# EPICS substitutions: db/MLout.substitutions
file "/epics/iocs/MachineLearn/db/MLout_sub.db"
{
pattern
{CELL, WIRE,  MODE}
{"01", "33", "lls"}
{"01", "34", "lls"}
{"01", "35", "lls"}
{"01", "36", "lls"}
{"01", "37", "lls"}
{"01", "38", "lls"}
{"01", "39", "lls"}
{"01", "40", "lls"}
{"01", "41", "lls"}
{"01", "42", "lls"}
{"01", "43", "lls"}
{"01", "44", "lls"}
{"01", "45", "lls"}
{"01", "46", "lls"}
{"01", "47", "lls"}
{"01", "48", "lls"}
{"01", "49", "lls"}
{"01", "50", "lls"}
{"01", "51", "lls"}
{"01", "52", "lls"}

{"02", "33", "lls"}
{"02", "34", "lls"}
{"02", "35", "lls"}
{"02", "36", "lls"}
{"02", "37", "lls"}
{"02", "38", "lls"}
{"02", "39", "lls"}
{"02", "40", "lls"}
{"02", "41", "lls"}
{"02", "42", "lls"}
{"02", "43", "lls"}
{"02", "44", "lls"}
{"02", "45", "lls"}
{"02", "46", "lls"}
{"02", "47", "lls"}
{"02", "48", "lls"}
{"02", "49", "lls"}
{"02", "50", "lls"}
{"02", "51", "lls"}
{"02", "52", "lls"}

{"03", "55", "lls"}
{"03", "56", "lls"}
{"03", "57", "lls"}
{"03", "58", "lls"}
{"03", "59", "lls"}
{"03", "60", "lls"}
{"03", "61", "lls"}
{"03", "62", "lls"}
{"03", "63", "lls"}
{"03", "64", "lls"}
{"03", "65", "lls"}
{"03", "66", "lls"}
{"03", "67", "lls"}
{"03", "68", "lls"}
{"03", "69", "lls"}
{"03", "70", "lls"}
{"03", "71", "lls"}
{"03", "72", "lls"}
{"03", "73", "lls"}
{"03", "74", "lls"}

{"04", "33", "lls"}
{"04", "34", "lls"}
{"04", "35", "lls"}
{"04", "36", "lls"}
{"04", "37", "lls"}
{"04", "38", "lls"}
{"04", "39", "lls"}
{"04", "40", "lls"}
{"04", "41", "lls"}
{"04", "42", "lls"}
{"04", "43", "lls"}
{"04", "44", "lls"}
{"04", "45", "lls"}
{"04", "46", "lls"}
{"04", "47", "lls"}
{"04", "48", "lls"}
{"04", "49", "lls"}
{"04", "50", "lls"}
{"04", "51", "lls"}
{"04", "52", "lls"}

{"05", "33", "lls"}
{"05", "34", "lls"}
{"05", "35", "lls"}
{"05", "36", "lls"}
{"05", "37", "lls"}
{"05", "38", "lls"}
{"05", "39", "lls"}
{"05", "40", "lls"}
{"05", "41", "lls"}
{"05", "42", "lls"}
{"05", "43", "lls"}
{"05", "44", "lls"}
{"05", "45", "lls"}
{"05", "46", "lls"}
{"05", "47", "lls"}
{"05", "48", "lls"}
{"05", "49", "lls"}
{"05", "50", "lls"}
{"05", "51", "lls"}
{"05", "52", "lls"}

{"06", "33", "lls"}
{"06", "34", "lls"}
{"06", "35", "lls"}
{"06", "36", "lls"}
{"06", "37", "lls"}
{"06", "38", "lls"}
{"06", "39", "lls"}
{"06", "40", "lls"}
{"06", "41", "lls"}
{"06", "42", "lls"}
{"06", "43", "lls"}
{"06", "44", "lls"}
{"06", "45", "lls"}
{"06", "46", "lls"}
{"06", "47", "lls"}
{"06", "48", "lls"}
{"06", "49", "lls"}
{"06", "50", "lls"}
{"06", "51", "lls"}
{"06", "52", "lls"}

{"07", "33", "lls"}
{"07", "34", "lls"}
{"07", "35", "lls"}
{"07", "36", "lls"}
{"07", "37", "lls"}
{"07", "38", "lls"}
{"07", "39", "lls"}
{"07", "40", "lls"}
{"07", "41", "lls"}
{"07", "42", "lls"}
{"07", "43", "lls"}
{"07", "44", "lls"}
{"07", "45", "lls"}
{"07", "46", "lls"}
{"07", "47", "lls"}
{"07", "48", "lls"}
{"07", "49", "lls"}
{"07", "50", "lls"}
{"07", "51", "lls"}
{"07", "52", "lls"}

{"08", "33", "lls"}
{"08", "34", "lls"}
{"08", "35", "lls"}
{"08", "36", "lls"}
{"08", "37", "lls"}
{"08", "38", "lls"}
{"08", "39", "lls"}
{"08", "40", "lls"}
{"08", "41", "lls"}
{"08", "42", "lls"}
{"08", "43", "lls"}
{"08", "44", "lls"}
{"08", "45", "lls"}
{"08", "46", "lls"}
{"08", "47", "lls"}
{"08", "48", "lls"}
{"08", "49", "lls"}
{"08", "50", "lls"}
{"08", "51", "lls"}
{"08", "52", "lls"}

{"09", "33", "lls"}
{"09", "34", "lls"}
{"09", "35", "lls"}
{"09", "36", "lls"}
{"09", "37", "lls"}
{"09", "38", "lls"}
{"09", "39", "lls"}
{"09", "40", "lls"}
{"09", "41", "lls"}
{"09", "42", "lls"}
{"09", "43", "lls"}
{"09", "44", "lls"}
{"09", "45", "lls"}
{"09", "46", "lls"}
{"09", "47", "lls"}
{"09", "48", "lls"}
{"09", "49", "lls"}
{"09", "50", "lls"}
{"09", "51", "lls"}
{"09", "52", "lls"}

{"10", "33", "lls"}
{"10", "34", "lls"}
{"10", "35", "lls"}
{"10", "36", "lls"}
{"10", "37", "lls"}
{"10", "38", "lls"}
{"10", "39", "lls"}
{"10", "40", "lls"}
{"10", "41", "lls"}
{"10", "42", "lls"}
{"10", "43", "lls"}
{"10", "44", "lls"}
{"10", "45", "lls"}
{"10", "46", "lls"}
{"10", "47", "lls"}
{"10", "48", "lls"}
{"10", "49", "lls"}
{"10", "50", "lls"}
{"10", "51", "lls"}
{"10", "52", "lls"}

{"11", "33", "lls"}
{"11", "34", "lls"}
{"11", "35", "lls"}
{"11", "36", "lls"}
{"11", "37", "lls"}
{"11", "38", "lls"}
{"11", "39", "lls"}
{"11", "40", "lls"}
{"11", "41", "lls"}
{"11", "42", "lls"}
{"11", "43", "lls"}
{"11", "44", "lls"}
{"11", "45", "lls"}
{"11", "46", "lls"}
{"11", "47", "lls"}
{"11", "48", "lls"}
{"11", "49", "lls"}
{"11", "50", "lls"}
{"11", "51", "lls"}
{"11", "52", "lls"}

{"12", "33", "lls"}
{"12", "34", "lls"}
{"12", "35", "lls"}
{"12", "36", "lls"}
{"12", "37", "lls"}
{"12", "38", "lls"}
{"12", "39", "lls"}
{"12", "40", "lls"}
{"12", "41", "lls"}
{"12", "42", "lls"}
{"12", "43", "lls"}
{"12", "44", "lls"}
{"12", "45", "lls"}
{"12", "46", "lls"}
{"12", "47", "lls"}
{"12", "48", "lls"}
{"12", "49", "lls"}
{"12", "50", "lls"}
{"12", "51", "lls"}
{"12", "52", "lls"}

{"13", "33", "lls"}
{"13", "34", "lls"}
{"13", "35", "lls"}
{"13", "36", "lls"}
{"13", "37", "lls"}
{"13", "38", "lls"}
{"13", "39", "lls"}
{"13", "40", "lls"}
{"13", "41", "lls"}
{"13", "42", "lls"}
{"13", "43", "lls"}
{"13", "44", "lls"}
{"13", "45", "lls"}
{"13", "46", "lls"}
{"13", "47", "lls"}
{"13", "48", "lls"}
{"13", "49", "lls"}
{"13", "50", "lls"}
{"13", "51", "lls"}
{"13", "52", "lls"}
{"13", "53", "lls"}
{"13", "54", "lls"}
{"13", "55", "lls"}
{"13", "56", "lls"}

{"14", "33", "lls"}
{"14", "34", "lls"}
{"14", "35", "lls"}
{"14", "36", "lls"}
{"14", "37", "lls"}
{"14", "38", "lls"}
{"14", "39", "lls"}
{"14", "40", "lls"}
{"14", "41", "lls"}
{"14", "42", "lls"}
{"14", "43", "lls"}
{"14", "44", "lls"}
{"14", "45", "lls"}
{"14", "46", "lls"}
{"14", "47", "lls"}
{"14", "48", "lls"}
{"14", "49", "lls"}
{"14", "50", "lls"}
{"14", "51", "lls"}
{"14", "52", "lls"}

{"15", "33", "lls"}
{"15", "34", "lls"}
{"15", "35", "lls"}
{"15", "36", "lls"}
{"15", "37", "lls"}
{"15", "38", "lls"}
{"15", "39", "lls"}
{"15", "40", "lls"}
{"15", "41", "lls"}
{"15", "42", "lls"}
{"15", "43", "lls"}
{"15", "44", "lls"}
{"15", "45", "lls"}
{"15", "46", "lls"}
{"15", "47", "lls"}
{"15", "48", "lls"}
{"15", "49", "lls"}
{"15", "50", "lls"}
{"15", "51", "lls"}
{"15", "52", "lls"}

{"16", "33", "lls"}
{"16", "34", "lls"}
{"16", "35", "lls"}
{"16", "36", "lls"}
{"16", "37", "lls"}
{"16", "38", "lls"}
{"16", "39", "lls"}
{"16", "40", "lls"}
{"16", "41", "lls"}
{"16", "42", "lls"}
{"16", "43", "lls"}
{"16", "44", "lls"}
{"16", "45", "lls"}
{"16", "46", "lls"}
{"16", "47", "lls"}
{"16", "48", "lls"}
{"16", "49", "lls"}
{"16", "50", "lls"}
{"16", "51", "lls"}
{"16", "52", "lls"}

{"17", "36", "lls"}
{"17", "37", "lls"}
{"17", "38", "lls"}
{"17", "39", "lls"}
{"17", "40", "lls"}
{"17", "41", "lls"}
{"17", "42", "lls"}
{"17", "43", "lls"}
{"17", "44", "lls"}
{"17", "45", "lls"}
{"17", "46", "lls"}
{"17", "47", "lls"}
{"17", "48", "lls"}
{"17", "49", "lls"}
{"17", "50", "lls"}
{"17", "51", "lls"}
{"17", "52", "lls"}
{"17", "53", "lls"}
{"17", "54", "lls"}
{"17", "55", "lls"}
{"17", "56", "lls"}
{"17", "57", "lls"}
{"17", "58", "lls"}
{"17", "59", "lls"}

{"18", "33", "lls"}
{"18", "34", "lls"}
{"18", "35", "lls"}
{"18", "36", "lls"}
{"18", "37", "lls"}
{"18", "38", "lls"}
{"18", "39", "lls"}
{"18", "40", "lls"}
{"18", "41", "lls"}
{"18", "42", "lls"}
{"18", "43", "lls"}
{"18", "44", "lls"}
{"18", "45", "lls"}
{"18", "46", "lls"}
{"18", "47", "lls"}
{"18", "48", "lls"}
{"18", "49", "lls"}
{"18", "50", "lls"}
{"18", "51", "lls"}
{"18", "52", "lls"}
{"18", "53", "lls"}
{"18", "54", "lls"}
{"18", "55", "lls"}
{"18", "56", "lls"}

{"19", "33", "lls"}
{"19", "34", "lls"}
{"19", "35", "lls"}
{"19", "36", "lls"}
{"19", "37", "lls"}
{"19", "38", "lls"}
{"19", "39", "lls"}
{"19", "40", "lls"}
{"19", "41", "lls"}
{"19", "42", "lls"}
{"19", "43", "lls"}
{"19", "44", "lls"}
{"19", "45", "lls"}
{"19", "46", "lls"}
{"19", "47", "lls"}
{"19", "48", "lls"}
{"19", "49", "lls"}
{"19", "50", "lls"}
{"19", "51", "lls"}
{"19", "52", "lls"}
{"19", "53", "lls"}
{"19", "54", "lls"}
{"19", "55", "lls"}
{"19", "56", "lls"}

{"20", "33", "lls"}
{"20", "34", "lls"}
{"20", "35", "lls"}
{"20", "36", "lls"}
{"20", "37", "lls"}
{"20", "38", "lls"}
{"20", "39", "lls"}
{"20", "40", "lls"}
{"20", "41", "lls"}
{"20", "42", "lls"}
{"20", "43", "lls"}
{"20", "44", "lls"}
{"20", "45", "lls"}
{"20", "46", "lls"}
{"20", "47", "lls"}
{"20", "48", "lls"}
{"20", "49", "lls"}
{"20", "50", "lls"}
{"20", "51", "lls"}
{"20", "52", "lls"}

{"21", "33", "lls"}
{"21", "34", "lls"}
{"21", "35", "lls"}
{"21", "36", "lls"}
{"21", "37", "lls"}
{"21", "38", "lls"}
{"21", "39", "lls"}
{"21", "40", "lls"}
{"21", "41", "lls"}
{"21", "42", "lls"}
{"21", "43", "lls"}
{"21", "44", "lls"}
{"21", "45", "lls"}
{"21", "46", "lls"}
{"21", "47", "lls"}
{"21", "48", "lls"}
{"21", "49", "lls"}
{"21", "50", "lls"}
{"21", "51", "lls"}
{"21", "52", "lls"}

{"22", "33", "lls"}
{"22", "34", "lls"}
{"22", "35", "lls"}
{"22", "36", "lls"}
{"22", "37", "lls"}
{"22", "38", "lls"}
{"22", "39", "lls"}
{"22", "40", "lls"}
{"22", "41", "lls"}
{"22", "42", "lls"}
{"22", "43", "lls"}
{"22", "44", "lls"}
{"22", "45", "lls"}
{"22", "46", "lls"}
{"22", "47", "lls"}
{"22", "48", "lls"}
{"22", "49", "lls"}
{"22", "50", "lls"}
{"22", "51", "lls"}
{"22", "52", "lls"}

{"23", "33", "lls"}
{"23", "34", "lls"}
{"23", "35", "lls"}
{"23", "36", "lls"}
{"23", "37", "lls"}
{"23", "38", "lls"}
{"23", "39", "lls"}
{"23", "40", "lls"}
{"23", "41", "lls"}
{"23", "42", "lls"}
{"23", "43", "lls"}
{"23", "44", "lls"}
{"23", "45", "lls"}
{"23", "46", "lls"}
{"23", "47", "lls"}
{"23", "48", "lls"}
{"23", "49", "lls"}
{"23", "50", "lls"}
{"23", "51", "lls"}
{"23", "52", "lls"}
{"23", "53", "lls"}
{"23", "54", "lls"}
{"23", "55", "lls"}
{"23", "56", "lls"}

{"24", "33", "lls"}
{"24", "34", "lls"}
{"24", "35", "lls"}
{"24", "36", "lls"}
{"24", "37", "lls"}
{"24", "38", "lls"}
{"24", "39", "lls"}
{"24", "40", "lls"}
{"24", "41", "lls"}
{"24", "42", "lls"}
{"24", "43", "lls"}
{"24", "44", "lls"}
{"24", "45", "lls"}
{"24", "46", "lls"}
{"24", "47", "lls"}
{"24", "48", "lls"}
{"24", "49", "lls"}
{"24", "50", "lls"}
{"24", "51", "lls"}
{"24", "52", "lls"}

{"25", "33", "lls"}
{"25", "34", "lls"}
{"25", "35", "lls"}
{"25", "36", "lls"}
{"25", "37", "lls"}
{"25", "38", "lls"}
{"25", "39", "lls"}
{"25", "40", "lls"}
{"25", "41", "lls"}
{"25", "42", "lls"}
{"25", "43", "lls"}
{"25", "44", "lls"}
{"25", "45", "lls"}
{"25", "46", "lls"}
{"25", "47", "lls"}
{"25", "48", "lls"}
{"25", "49", "lls"}
{"25", "50", "lls"}
{"25", "51", "lls"}
{"25", "52", "lls"}

{"26", "33", "lls"}
{"26", "34", "lls"}
{"26", "35", "lls"}
{"26", "36", "lls"}
{"26", "37", "lls"}
{"26", "38", "lls"}
{"26", "39", "lls"}
{"26", "40", "lls"}
{"26", "41", "lls"}
{"26", "42", "lls"}
{"26", "43", "lls"}
{"26", "44", "lls"}
{"26", "45", "lls"}
{"26", "46", "lls"}
{"26", "47", "lls"}
{"26", "48", "lls"}
{"26", "49", "lls"}
{"26", "50", "lls"}
{"26", "51", "lls"}
{"26", "52", "lls"}

{"27", "33", "lls"}
{"27", "34", "lls"}
{"27", "35", "lls"}
{"27", "36", "lls"}
{"27", "37", "lls"}
{"27", "38", "lls"}
{"27", "39", "lls"}
{"27", "40", "lls"}
{"27", "41", "lls"}
{"27", "42", "lls"}
{"27", "43", "lls"}
{"27", "44", "lls"}
{"27", "45", "lls"}
{"27", "46", "lls"}
{"27", "47", "lls"}
{"27", "48", "lls"}
{"27", "49", "lls"}
{"27", "50", "lls"}
{"27", "51", "lls"}
{"27", "52", "lls"}

{"28", "33", "lls"}
{"28", "34", "lls"}
{"28", "35", "lls"}
{"28", "36", "lls"}
{"28", "37", "lls"}
{"28", "38", "lls"}
{"28", "39", "lls"}
{"28", "40", "lls"}
{"28", "41", "lls"}
{"28", "42", "lls"}
{"28", "43", "lls"}
{"28", "44", "lls"}
{"28", "45", "lls"}
{"28", "46", "lls"}
{"28", "47", "lls"}
{"28", "48", "lls"}
{"28", "49", "lls"}
{"28", "50", "lls"}
{"28", "51", "lls"}
{"28", "52", "lls"}

{"29", "33", "lls"}
{"29", "34", "lls"}
{"29", "35", "lls"}
{"29", "36", "lls"}
{"29", "37", "lls"}
{"29", "38", "lls"}
{"29", "39", "lls"}
{"29", "40", "lls"}
{"29", "41", "lls"}
{"29", "42", "lls"}
{"29", "43", "lls"}
{"29", "44", "lls"}
{"29", "45", "lls"}
{"29", "46", "lls"}
{"29", "47", "lls"}
{"29", "48", "lls"}
{"29", "49", "lls"}
{"29", "50", "lls"}
{"29", "51", "lls"}
{"29", "52", "lls"}

{"30", "33", "lls"}
{"30", "34", "lls"}
{"30", "35", "lls"}
{"30", "36", "lls"}
{"30", "37", "lls"}
{"30", "38", "lls"}
{"30", "39", "lls"}
{"30", "40", "lls"}
{"30", "41", "lls"}
{"30", "42", "lls"}
{"30", "43", "lls"}
{"30", "44", "lls"}
{"30", "45", "lls"}
{"30", "46", "lls"}
{"30", "47", "lls"}
{"30", "48", "lls"}
{"30", "49", "lls"}
{"30", "50", "lls"}
{"30", "51", "lls"}
{"30", "52", "lls"}
}
